(*********************************** G.D S.p.A. - Technical Department ***********************************
============= PROGRAM INFO ============
FOLDER:             TBD
MACHINES INVOLVED:  TBD 

============= DESCRIPTION =============
csp machine declaration

============= REVISIONS ===============
Date		Version	 	Author      	Description             
----------	-------		------------  	--------------------------------------------
2019/04/05 	0000.00	 	M.Grasso		Creation of the PRG

**********************************************************************************************************)
(*$R process_ref := prc; $*)
PROGRAM csp_case_fc_os_lower
VAR
	
	prc:											process;
	prc_path:										STRING;
	
END_VAR

_read_var_input();

_object_manager();

IF NOT objects_running()
THEN
	RETURN;	
END_IF

_read_process_image();

_mode_manager();

_set_runtime_properties();

(********************************* BODY *********************************)
(************************************************************************)

_handle_messages();

_write_output();

ACTION _handle_messages:
;
END_ACTION

ACTION _handle_process_test:
;
END_ACTION

ACTION _mode_manager:
IF process_mode_req_is_pending(prc)
THEN
    process_apply_mode_req_first_step(prc);
    CASE process_get_mode(prc) OF
        MODE_TO_ABSENT:
			;
        MODE_TO_INACTIVE:
			;
        MODE_TO_TEST:
			;
        MODE_TO_OPERATIONAL:
			;
    END_CASE
    process_apply_mode_req_second_step(prc);
END_IF
END_ACTION

ACTION _object_manager:
IF objects_initialization()
THEN
	sub_process_init(
		object_name					:= 'csp_case_fc_os_lower.prc', 
		process						:= csp_case_flapControl_os.prc, 
		CONVERSION_this				:= prc);
		
	prc_path 						:= process_get_path(prc);
END_IF

IF objects_running()
THEN
	process_cycle(prc);
END_IF
END_ACTION

ACTION _read_process_image:
;
END_ACTION

ACTION _read_var_input:
;
END_ACTION

ACTION _set_runtime_properties:
;
END_ACTION

ACTION _write_output:
;
END_ACTION

END_PROGRAM

(* stored: Version 1.1.0.1, ProductVersion 3.1.4022.12
   POU csp_case_fc_os_lower: Id {7cf109b4-6939-41af-aafd-a2167448cc0f}, SpecialFunc None
   Action _handle_messages: Id {2e7f0bde-8996-41ed-ad79-c89a859cbc6b}
   Action _handle_process_test: Id {aadba697-25e5-4b17-984f-3a04d45f470c}
   Action _mode_manager: Id {9007a339-fa41-4807-a5b2-36b1f9fe07b4}
   Action _object_manager: Id {948d5b28-4c19-43f4-88de-b5386e35fe0f}
   Action _read_process_image: Id {1b77a763-f166-4f2f-bf2b-3a2c22ae3188}
   Action _read_var_input: Id {f69f3dad-76e4-47c5-abc1-4e986deeff16}
   Action _set_runtime_properties: Id {b8dd4be7-5016-43db-aa90-c3947984b83e}
   Action _write_output: Id {d3f82fed-5a17-44b8-b2ff-ce68d7650997} *)
